TYPE SmokeControlParameters :
STRUCT
	MidiSmoke: MidiSmokeParameters;
	DamperModules: SxDuoParameters;
END_STRUCT
END_TYPE

(* stored: Version 1.1.0.1, ProductVersion 3.1.4024.6
   DUT SmokeControlParameters: Id {006331c9-eeba-45a1-91ab-17ad59f5dd21} *)
